TYPE RegexMatch :
STRUCT
	found : BOOL;
	start : INT;
	length : INT;
	text : STRING;
END_STRUCT
END_TYPE

(* stored: Version 1.1.0.1, ProductVersion 3.1.4024.11
   DUT RegexMatch: Id {7ddf576e-ed24-4ed7-a56f-36fa1d4f7aa5} *)
